TYPE T_BCD_Status :
STRUCT
	/// Socket connected
	bolSocketConnected: BOOL;
	bolComChecked: BOOL;
END_STRUCT
END_TYPE

(* stored: Version 1.1.0.1, ProductVersion 3.1.0.26
   DUT T_BCD_Status: Id {b917762c-531c-47d1-904c-a37d4358f834} *)
